PROGRAM P_Demo_FB_JsonDomParser_ParseDocument
VAR
    fbParser : FB_JsonDomParser; // 父 FB 实例
    sJson : STRING(255);
    vRet : SJsonValue; // 返回值监视
    bTrigger : BOOL := FALSE; // 在线置 TRUE 触发一次调用
    bTriggerPrev : BOOL;
END_VAR

// =============================================================================
// 场景：接收一帧 MQTT JSON 报文，加载到 DOM 准备后续 Find / Get 操作。
// 价值：同步单次调用，调用后立刻可访问；省去维护 SAX 状态机的复杂度。
// 验证：登录 PLC 在线写 bTrigger := TRUE 触发，monitor 返回值/输出参数。具体步骤见下方注释。
// 验证步骤：
//   1. 右键 PLC 项目下 POUs 文件夹 → Add → Existing Item → 选本 .TcPOU 文件
//   2. 引用 Tc3_JsonXml（References → Add library）
//   3. 编译 → 登录 → 运行；按 verify 注释里给出的在线写值操作
// =============================================================================

// 上升沿触发一次方法调用并观察输出。
IF bTrigger AND NOT bTriggerPrev THEN
    vRet := fbParser.ParseDocument(
        sJson := sJson
    );
END_IF;
bTriggerPrev := bTrigger;

END_PROGRAM

(* stored: Version 1.1.0.1, ProductVersion 3.1.4024.5
   POU P_Demo_FB_JsonDomParser_ParseDocument: Id {1cfdbb49-095c-5bd1-b148-0e57e3d71541}, SpecialFunc None *)
